// TIA Portal V17 export
// export: Created 2025-06-26T07:49:16.300104Z, ExportSetting WithDefaults, DisplayName Totally Integrated Automation Portal, DisplayVersion V17 Update 8, DisplayName TIA Portal Openness, DisplayVersion V17 Update 8, DisplayName TIA Portal Version Control Interface, DisplayVersion V17, DisplayName STEP 7 Professional, DisplayVersion V17 Update 8, DisplayName STEP 7 Safety, DisplayVersion V17 Update 6, DisplayName WinCC Advanced, DisplayVersion V17 Update 8
FUNCTION_BLOCK "PumaInputProcessing"   // FB5, FBD
{ S7_Optimized_Access := 'TRUE' }
AUTHOR : Heaten
VERSION : 0.1
// stored: AutoNumber true, IsIECCheckEnabled false, IsRetainMemResEnabled false, MemoryReserve 0, SetENOAutomatically false, UDAEnableTagReadback false
   VAR_INPUT
      bEnable : Bool;
   END_VAR
   VAR
      Dummy : Bool;
   END_VAR
   VAR_TEMP
      bCommOk : Bool;   // Puma is running
      fDummy : Real;
   END_VAR
BEGIN

REGION Network 1: Comm ok
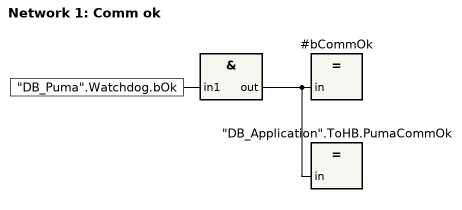
   #bCommOk := "DB_Puma".Watchdog.bOk;
   "DB_Application".ToHB.PumaCommOk := "DB_Puma".Watchdog.bOk;
END_REGION

REGION Network 2: Test Support System values (AI)
   // TSS = Test Support System
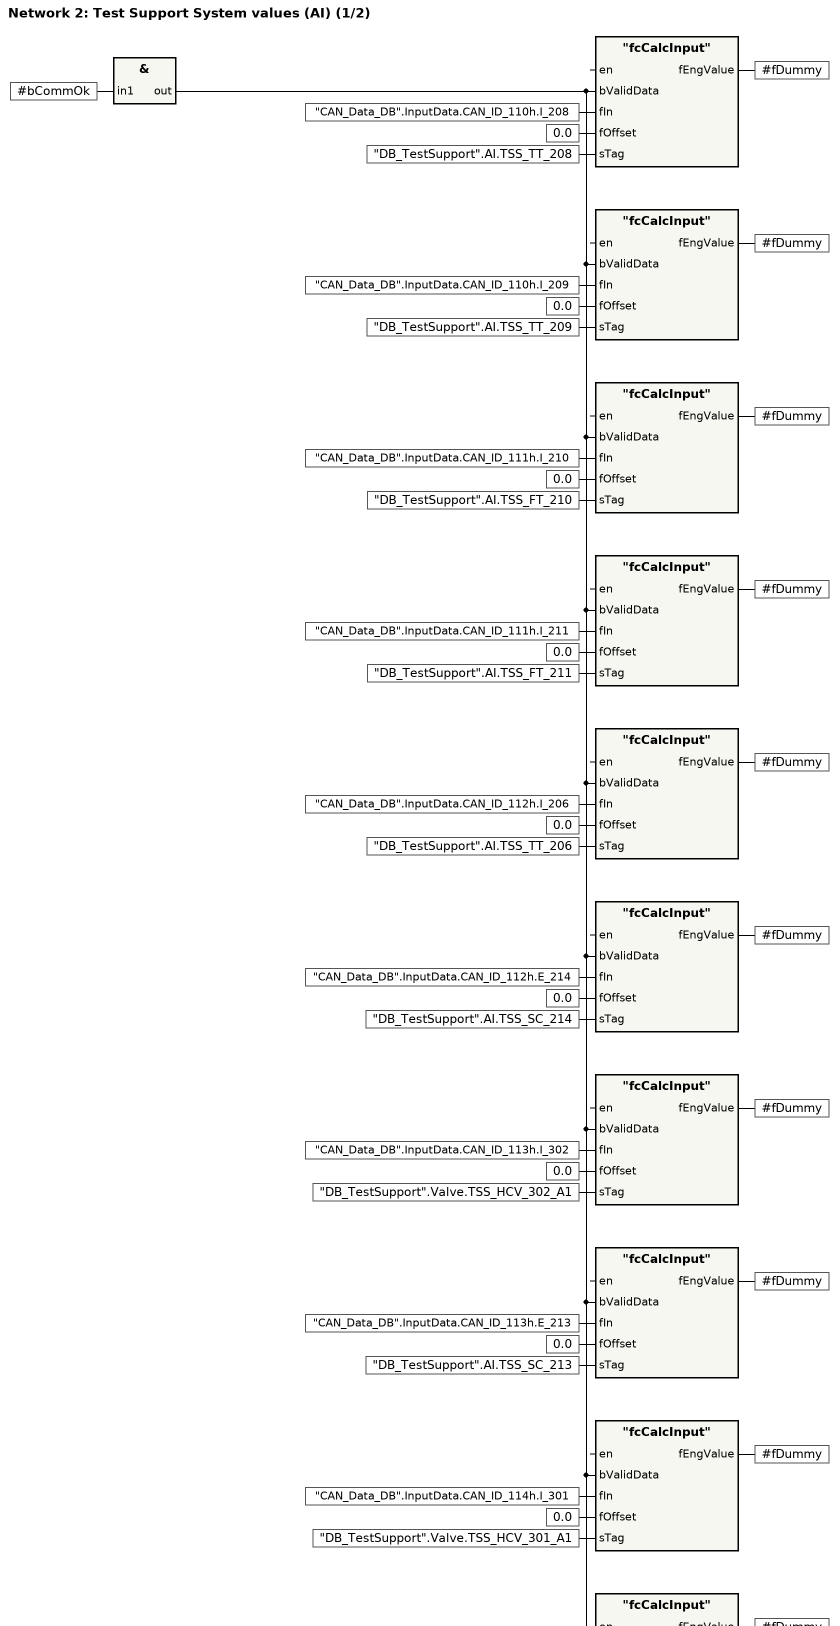
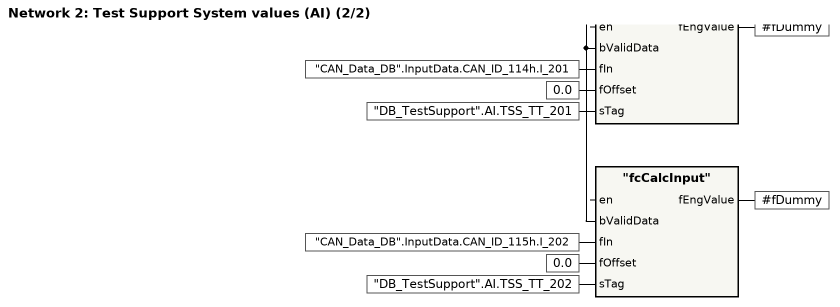
   "fcCalcInput"(bValidData := #bCommOk,
                 fIn := "CAN_Data_DB".InputData.CAN_ID_110h.I_208,
                 fOffset := 0.0,
                 sTag := "DB_TestSupport".AI.TSS_TT_208,
                 fEngValue => #fDummy);
   "fcCalcInput"(bValidData := #bCommOk,
                 fIn := "CAN_Data_DB".InputData.CAN_ID_110h.I_209,
                 fOffset := 0.0,
                 sTag := "DB_TestSupport".AI.TSS_TT_209,
                 fEngValue => #fDummy);
   "fcCalcInput"(bValidData := #bCommOk,
                 fIn := "CAN_Data_DB".InputData.CAN_ID_111h.I_210,
                 fOffset := 0.0,
                 sTag := "DB_TestSupport".AI.TSS_FT_210,
                 fEngValue => #fDummy);
   "fcCalcInput"(bValidData := #bCommOk,
                 fIn := "CAN_Data_DB".InputData.CAN_ID_111h.I_211,
                 fOffset := 0.0,
                 sTag := "DB_TestSupport".AI.TSS_FT_211,
                 fEngValue => #fDummy);
   "fcCalcInput"(bValidData := #bCommOk,
                 fIn := "CAN_Data_DB".InputData.CAN_ID_112h.I_206,
                 fOffset := 0.0,
                 sTag := "DB_TestSupport".AI.TSS_TT_206,
                 fEngValue => #fDummy);
   "fcCalcInput"(bValidData := #bCommOk,
                 fIn := "CAN_Data_DB".InputData.CAN_ID_112h.E_214,
                 fOffset := 0.0,
                 sTag := "DB_TestSupport".AI.TSS_SC_214,
                 fEngValue => #fDummy);
   "fcCalcInput"(bValidData := #bCommOk,
                 fIn := "CAN_Data_DB".InputData.CAN_ID_113h.I_302,
                 fOffset := 0.0,
                 sTag := "DB_TestSupport".Valve.TSS_HCV_302_A1,
                 fEngValue => #fDummy);
   "fcCalcInput"(bValidData := #bCommOk,
                 fIn := "CAN_Data_DB".InputData.CAN_ID_113h.E_213,
                 fOffset := 0.0,
                 sTag := "DB_TestSupport".AI.TSS_SC_213,
                 fEngValue => #fDummy);
   "fcCalcInput"(bValidData := #bCommOk,
                 fIn := "CAN_Data_DB".InputData.CAN_ID_114h.I_301,
                 fOffset := 0.0,
                 sTag := "DB_TestSupport".Valve.TSS_HCV_301_A1,
                 fEngValue => #fDummy);
   "fcCalcInput"(bValidData := #bCommOk,
                 fIn := "CAN_Data_DB".InputData.CAN_ID_114h.I_201,
                 fOffset := 0.0,
                 sTag := "DB_TestSupport".AI.TSS_TT_201,
                 fEngValue => #fDummy);
   "fcCalcInput"(bValidData := #bCommOk,
                 fIn := "CAN_Data_DB".InputData.CAN_ID_115h.I_202,
                 fOffset := 0.0,
                 sTag := "DB_TestSupport".AI.TSS_TT_202,
                 fEngValue => #fDummy);
END_REGION

REGION Network 3: Steam Adapter values (AI)
   // TSA = TSS Steam Adapters
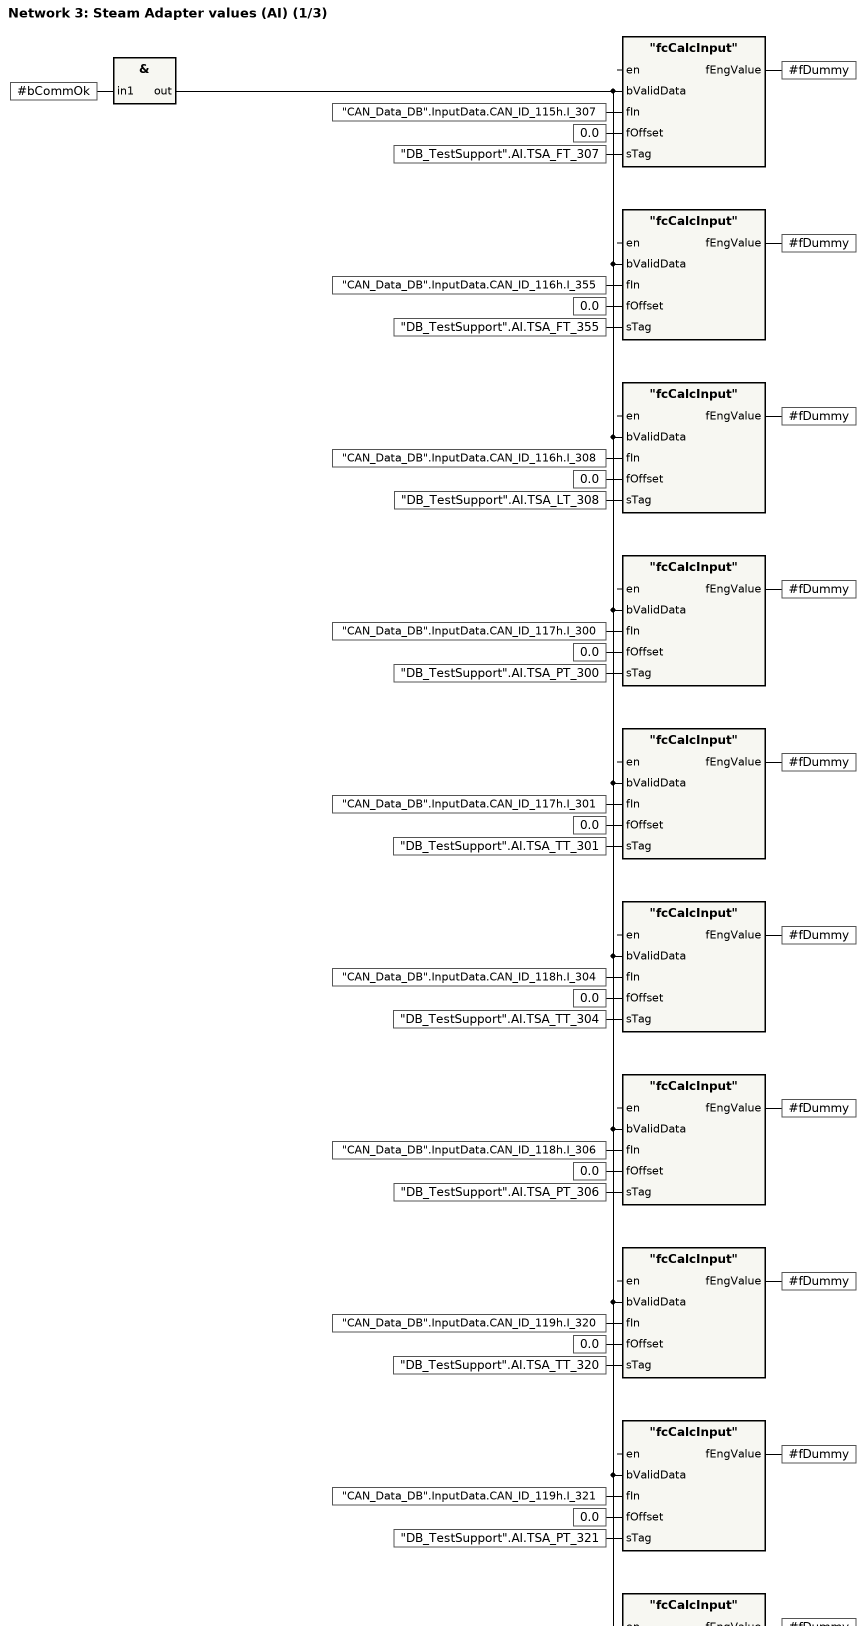
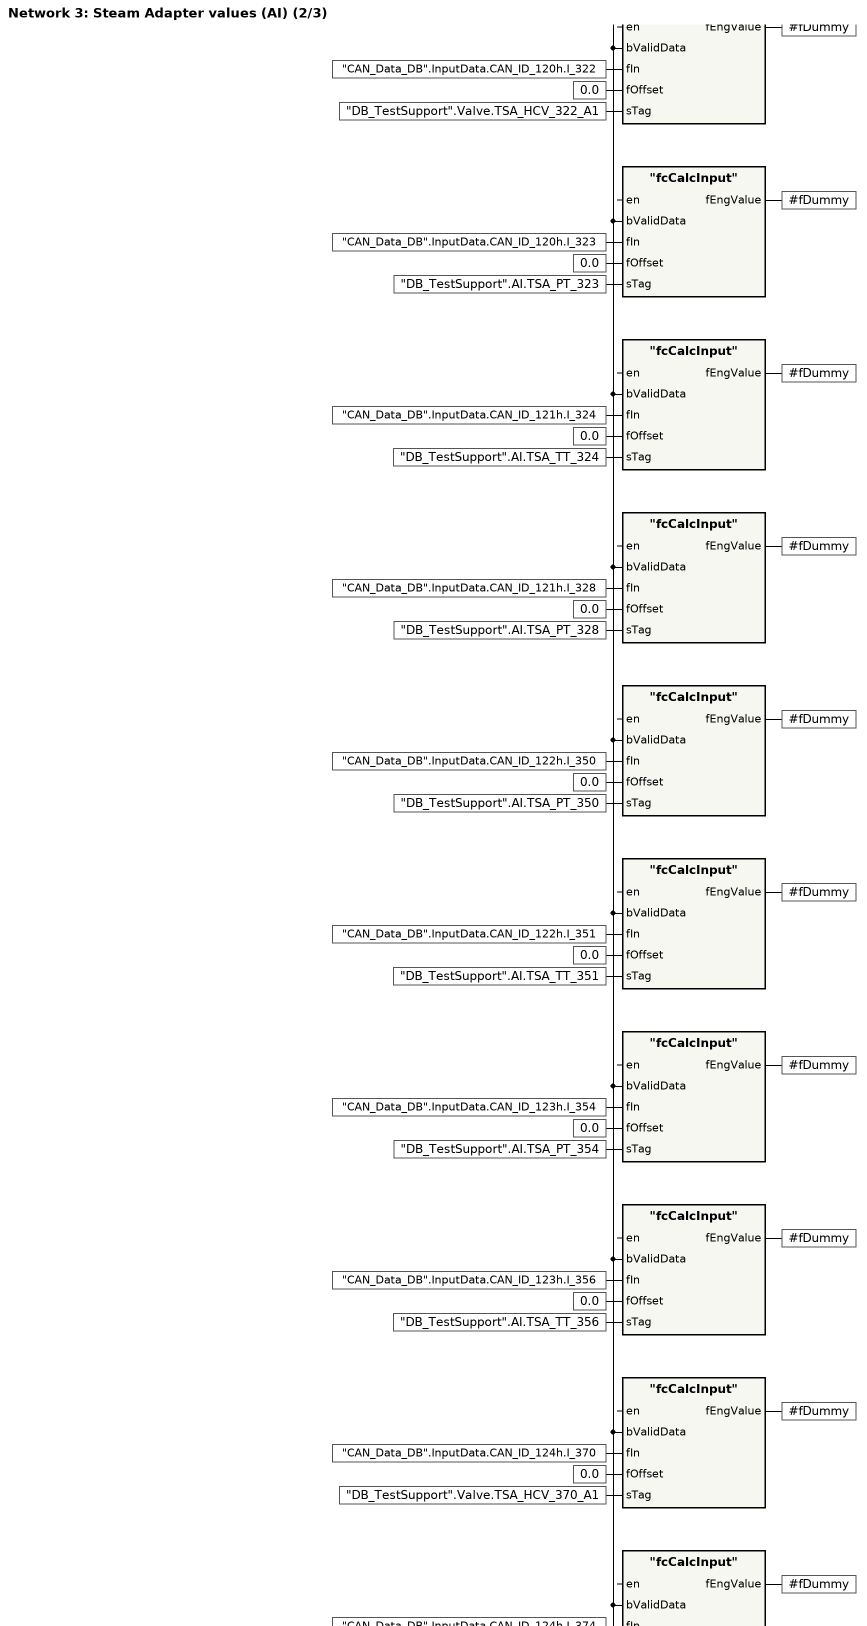
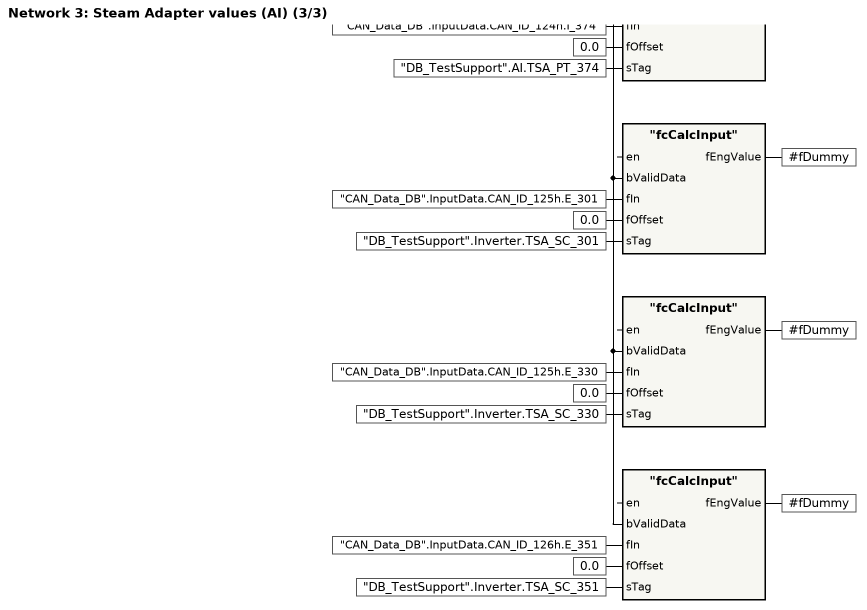
   "fcCalcInput"(bValidData := #bCommOk,
                 fIn := "CAN_Data_DB".InputData.CAN_ID_115h.I_307,
                 fOffset := 0.0,
                 sTag := "DB_TestSupport".AI.TSA_FT_307,
                 fEngValue => #fDummy);
   "fcCalcInput"(bValidData := #bCommOk,
                 fIn := "CAN_Data_DB".InputData.CAN_ID_116h.I_355,
                 fOffset := 0.0,
                 sTag := "DB_TestSupport".AI.TSA_FT_355,
                 fEngValue => #fDummy);
   "fcCalcInput"(bValidData := #bCommOk,
                 fIn := "CAN_Data_DB".InputData.CAN_ID_116h.I_308,
                 fOffset := 0.0,
                 sTag := "DB_TestSupport".AI.TSA_LT_308,
                 fEngValue => #fDummy);
   "fcCalcInput"(bValidData := #bCommOk,
                 fIn := "CAN_Data_DB".InputData.CAN_ID_117h.I_300,
                 fOffset := 0.0,
                 sTag := "DB_TestSupport".AI.TSA_PT_300,
                 fEngValue => #fDummy);
   "fcCalcInput"(bValidData := #bCommOk,
                 fIn := "CAN_Data_DB".InputData.CAN_ID_117h.I_301,
                 fOffset := 0.0,
                 sTag := "DB_TestSupport".AI.TSA_TT_301,
                 fEngValue => #fDummy);
   "fcCalcInput"(bValidData := #bCommOk,
                 fIn := "CAN_Data_DB".InputData.CAN_ID_118h.I_304,
                 fOffset := 0.0,
                 sTag := "DB_TestSupport".AI.TSA_TT_304,
                 fEngValue => #fDummy);
   "fcCalcInput"(bValidData := #bCommOk,
                 fIn := "CAN_Data_DB".InputData.CAN_ID_118h.I_306,
                 fOffset := 0.0,
                 sTag := "DB_TestSupport".AI.TSA_PT_306,
                 fEngValue => #fDummy);
   "fcCalcInput"(bValidData := #bCommOk,
                 fIn := "CAN_Data_DB".InputData.CAN_ID_119h.I_320,
                 fOffset := 0.0,
                 sTag := "DB_TestSupport".AI.TSA_TT_320,
                 fEngValue => #fDummy);
   "fcCalcInput"(bValidData := #bCommOk,
                 fIn := "CAN_Data_DB".InputData.CAN_ID_119h.I_321,
                 fOffset := 0.0,
                 sTag := "DB_TestSupport".AI.TSA_PT_321,
                 fEngValue => #fDummy);
   "fcCalcInput"(bValidData := #bCommOk,
                 fIn := "CAN_Data_DB".InputData.CAN_ID_120h.I_322,
                 fOffset := 0.0,
                 sTag := "DB_TestSupport".Valve.TSA_HCV_322_A1,
                 fEngValue => #fDummy);
   "fcCalcInput"(bValidData := #bCommOk,
                 fIn := "CAN_Data_DB".InputData.CAN_ID_120h.I_323,
                 fOffset := 0.0,
                 sTag := "DB_TestSupport".AI.TSA_PT_323,
                 fEngValue => #fDummy);
   "fcCalcInput"(bValidData := #bCommOk,
                 fIn := "CAN_Data_DB".InputData.CAN_ID_121h.I_324,
                 fOffset := 0.0,
                 sTag := "DB_TestSupport".AI.TSA_TT_324,
                 fEngValue => #fDummy);
   "fcCalcInput"(bValidData := #bCommOk,
                 fIn := "CAN_Data_DB".InputData.CAN_ID_121h.I_328,
                 fOffset := 0.0,
                 sTag := "DB_TestSupport".AI.TSA_PT_328,
                 fEngValue => #fDummy);
   "fcCalcInput"(bValidData := #bCommOk,
                 fIn := "CAN_Data_DB".InputData.CAN_ID_122h.I_350,
                 fOffset := 0.0,
                 sTag := "DB_TestSupport".AI.TSA_PT_350,
                 fEngValue => #fDummy);
   "fcCalcInput"(bValidData := #bCommOk,
                 fIn := "CAN_Data_DB".InputData.CAN_ID_122h.I_351,
                 fOffset := 0.0,
                 sTag := "DB_TestSupport".AI.TSA_TT_351,
                 fEngValue => #fDummy);
   "fcCalcInput"(bValidData := #bCommOk,
                 fIn := "CAN_Data_DB".InputData.CAN_ID_123h.I_354,
                 fOffset := 0.0,
                 sTag := "DB_TestSupport".AI.TSA_PT_354,
                 fEngValue => #fDummy);
   "fcCalcInput"(bValidData := #bCommOk,
                 fIn := "CAN_Data_DB".InputData.CAN_ID_123h.I_356,
                 fOffset := 0.0,
                 sTag := "DB_TestSupport".AI.TSA_TT_356,
                 fEngValue => #fDummy);
   "fcCalcInput"(bValidData := #bCommOk,
                 fIn := "CAN_Data_DB".InputData.CAN_ID_124h.I_370,
                 fOffset := 0.0,
                 sTag := "DB_TestSupport".Valve.TSA_HCV_370_A1,
                 fEngValue => #fDummy);
   "fcCalcInput"(bValidData := #bCommOk,
                 fIn := "CAN_Data_DB".InputData.CAN_ID_124h.I_374,
                 fOffset := 0.0,
                 sTag := "DB_TestSupport".AI.TSA_PT_374,
                 fEngValue => #fDummy);
   "fcCalcInput"(bValidData := #bCommOk,
                 fIn := "CAN_Data_DB".InputData.CAN_ID_125h.E_301,
                 fOffset := 0.0,
                 sTag := "DB_TestSupport".Inverter.TSA_SC_301,
                 fEngValue => #fDummy);
   "fcCalcInput"(bValidData := #bCommOk,
                 fIn := "CAN_Data_DB".InputData.CAN_ID_125h.E_330,
                 fOffset := 0.0,
                 sTag := "DB_TestSupport".Inverter.TSA_SC_330,
                 fEngValue => #fDummy);
   "fcCalcInput"(bValidData := #bCommOk,
                 fIn := "CAN_Data_DB".InputData.CAN_ID_126h.E_351,
                 fOffset := 0.0,
                 sTag := "DB_TestSupport".Inverter.TSA_SC_351,
                 fEngValue => #fDummy);
END_REGION

REGION Network 4: Steam Adapter values (DI)
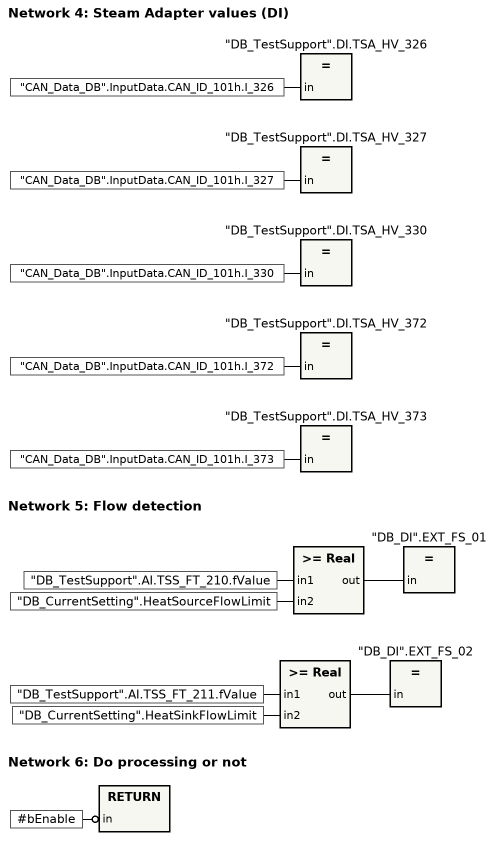
   "DB_TestSupport".DI.TSA_HV_326 := "CAN_Data_DB".InputData.CAN_ID_101h.I_326;
   "DB_TestSupport".DI.TSA_HV_327 := "CAN_Data_DB".InputData.CAN_ID_101h.I_327;
   "DB_TestSupport".DI.TSA_HV_330 := "CAN_Data_DB".InputData.CAN_ID_101h.I_330;
   "DB_TestSupport".DI.TSA_HV_372 := "CAN_Data_DB".InputData.CAN_ID_101h.I_372;
   "DB_TestSupport".DI.TSA_HV_373 := "CAN_Data_DB".InputData.CAN_ID_101h.I_373;
END_REGION

REGION Network 5: Flow detection
   "DB_DI".EXT_FS_01 := "DB_TestSupport".AI.TSS_FT_210.fValue >= "DB_CurrentSetting".HeatSourceFlowLimit;
   "DB_DI".EXT_FS_02 := "DB_TestSupport".AI.TSS_FT_211.fValue >= "DB_CurrentSetting".HeatSinkFlowLimit;
END_REGION

REGION Network 6: Do processing or not
   IF NOT #bEnable THEN
       ENO := TRUE;
       RETURN;
   END_IF;
END_REGION
END_FUNCTION_BLOCK
